// TIA Portal V19 export
FUNCTION "KP8 Interface" : Void   // FC3, LAD
{ S7_Optimized_Access := 'TRUE' }
// stored: SetENOAutomatically false
   VAR_TEMP
      RetVal : Int;
   END_VAR
   VAR_TEMP   // added for the SCL form of the ladder/FBD networks
      _w1 : Bool;
      _w2 : Bool;
   END_VAR
BEGIN

REGION Network 1: Turn all buttons white by default
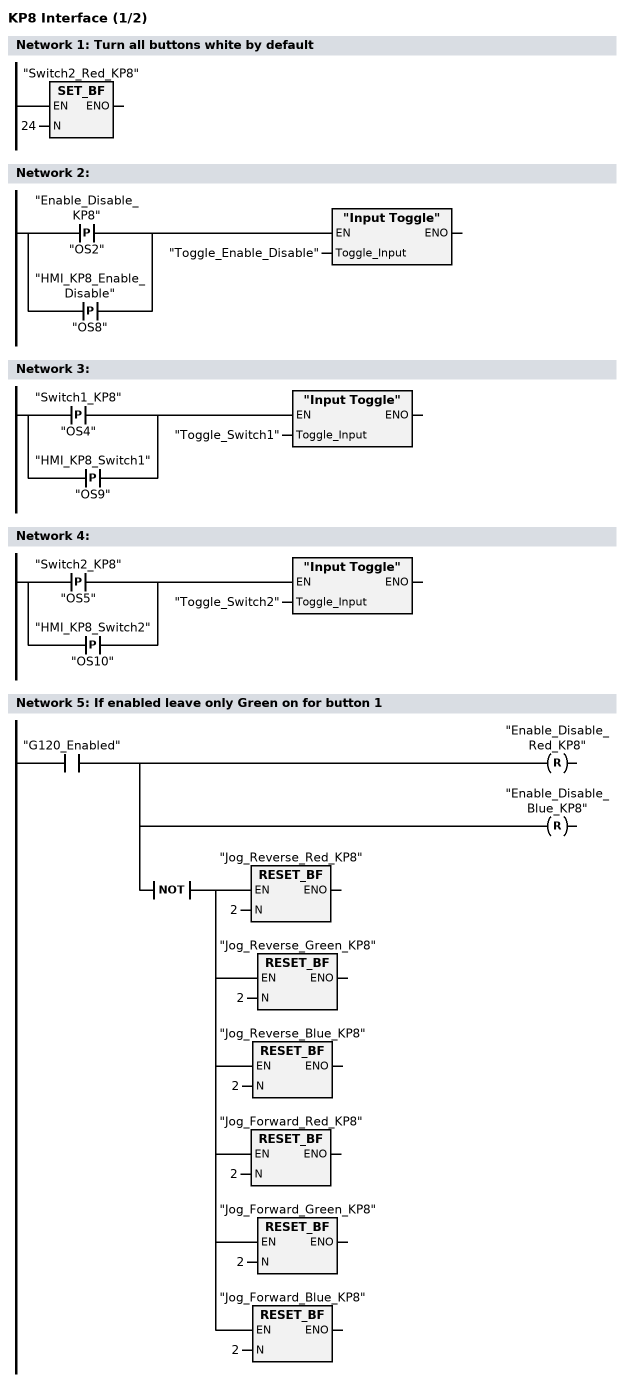
   // no SCL statement known for SBitfield: written as a call
   SET_BF(operand := "Switch2_Red_KP8", n := 24);
END_REGION

REGION Network 2
   RUNG wire#powerrail
      P_Contact(operand := "Enable_Disable_KP8", bit := "OS2")
      wire#w1
      "Input Toggle"(Toggle_Input := "Toggle_Enable_Disable")
   END_RUNG
   RUNG wire#powerrail
      P_Contact(operand := "HMI_KP8_Enable_Disable", bit := "OS8")
   END_RUNG wire#w1
   // the same network as SCL:
   #_w1 := "Enable_Disable_KP8" AND NOT "OS2";   // rising edge of "Enable_Disable_KP8"
   "OS2" := "Enable_Disable_KP8";
   #_w2 := "HMI_KP8_Enable_Disable" AND NOT "OS8";   // rising edge of "HMI_KP8_Enable_Disable"
   "OS8" := "HMI_KP8_Enable_Disable";
   IF #_w1 OR #_w2 THEN "Input Toggle"(Toggle_Input := "Toggle_Enable_Disable"); END_IF;
END_REGION

REGION Network 3
   RUNG wire#powerrail
      P_Contact(operand := "Switch1_KP8", bit := "OS4")
      wire#w1
      "Input Toggle"(Toggle_Input := "Toggle_Switch1")
   END_RUNG
   RUNG wire#powerrail
      P_Contact(operand := "HMI_KP8_Switch1", bit := "OS9")
   END_RUNG wire#w1
   // the same network as SCL:
   #_w1 := "Switch1_KP8" AND NOT "OS4";   // rising edge of "Switch1_KP8"
   "OS4" := "Switch1_KP8";
   #_w2 := "HMI_KP8_Switch1" AND NOT "OS9";   // rising edge of "HMI_KP8_Switch1"
   "OS9" := "HMI_KP8_Switch1";
   IF #_w1 OR #_w2 THEN "Input Toggle"(Toggle_Input := "Toggle_Switch1"); END_IF;
END_REGION

REGION Network 4
   RUNG wire#powerrail
      P_Contact(operand := "Switch2_KP8", bit := "OS5")
      wire#w1
      "Input Toggle"(Toggle_Input := "Toggle_Switch2")
   END_RUNG
   RUNG wire#powerrail
      P_Contact(operand := "HMI_KP8_Switch2", bit := "OS10")
   END_RUNG wire#w1
   // the same network as SCL:
   #_w1 := "Switch2_KP8" AND NOT "OS5";   // rising edge of "Switch2_KP8"
   "OS5" := "Switch2_KP8";
   #_w2 := "HMI_KP8_Switch2" AND NOT "OS10";   // rising edge of "HMI_KP8_Switch2"
   "OS10" := "HMI_KP8_Switch2";
   IF #_w1 OR #_w2 THEN "Input Toggle"(Toggle_Input := "Toggle_Switch2"); END_IF;
END_REGION

REGION Network 5: If enabled leave only Green on for button 1
   // no SCL statement known for RBitfield: written as a call
   IF "G120_Enabled" THEN
       "Enable_Disable_Red_KP8" := FALSE;
       "Enable_Disable_Blue_KP8" := FALSE;
   END_IF;
   #_w1 := NOT "G120_Enabled";
   IF #_w1 THEN
       RESET_BF(operand := "Jog_Reverse_Red_KP8", n := 2);
       RESET_BF(operand := "Jog_Reverse_Green_KP8", n := 2);
       RESET_BF(operand := "Jog_Reverse_Blue_KP8", n := 2);
       RESET_BF(operand := "Jog_Forward_Red_KP8", n := 2);
       RESET_BF(operand := "Jog_Forward_Green_KP8", n := 2);
       RESET_BF(operand := "Jog_Forward_Blue_KP8", n := 2);
   END_IF;
END_REGION

REGION Network 6: If there is an error flash red for button 5 by turning off other 2 leds
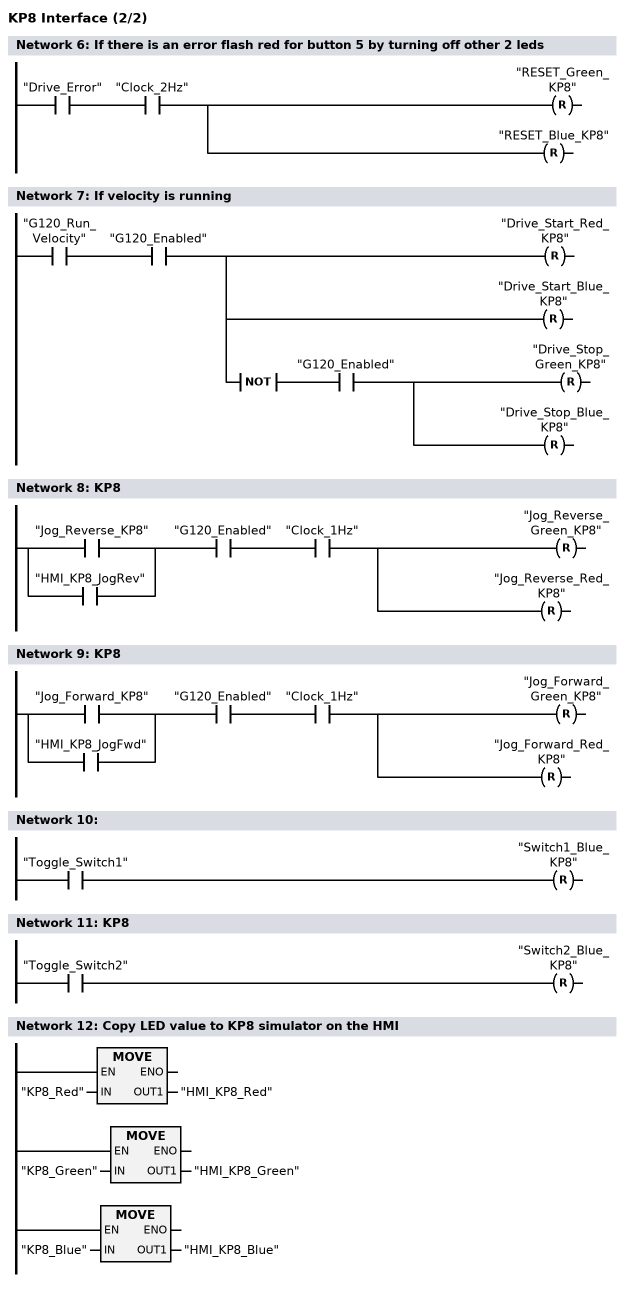
   RUNG wire#powerrail
      Contact( "Drive_Error" )
      Contact( "Clock_2Hz" )
      wire#w1
      R_Coil( "RESET_Green_KP8" )
   END_RUNG
   RUNG wire#w1
      R_Coil( "RESET_Blue_KP8" )
   END_RUNG
   // the same network as SCL:
   IF "Drive_Error" AND "Clock_2Hz" THEN
       "RESET_Green_KP8" := FALSE;
       "RESET_Blue_KP8" := FALSE;
   END_IF;
END_REGION

REGION Network 7: If velocity is running
   RUNG wire#powerrail
      Contact( "G120_Run_Velocity" )
      Contact( "G120_Enabled" )
      wire#w1
      R_Coil( "Drive_Start_Red_KP8" )
   END_RUNG
   RUNG wire#w1
      R_Coil( "Drive_Start_Blue_KP8" )
   END_RUNG
   RUNG wire#w1
      Not()
      Contact( "G120_Enabled" )
      wire#w2
      R_Coil( "Drive_Stop_Green_KP8" )
   END_RUNG
   RUNG wire#w2
      R_Coil( "Drive_Stop_Blue_KP8" )
   END_RUNG
   // the same network as SCL:
   #_w1 := "G120_Run_Velocity" AND "G120_Enabled";
   IF #_w1 THEN
       "Drive_Start_Red_KP8" := FALSE;
       "Drive_Start_Blue_KP8" := FALSE;
   END_IF;
   IF NOT #_w1 AND "G120_Enabled" THEN
       "Drive_Stop_Green_KP8" := FALSE;
       "Drive_Stop_Blue_KP8" := FALSE;
   END_IF;
END_REGION

REGION Network 8: KP8
   RUNG wire#powerrail
      Contact( "Jog_Reverse_KP8" )
      wire#w1
      Contact( "G120_Enabled" )
      Contact( "Clock_1Hz" )
      wire#w2
      R_Coil( "Jog_Reverse_Green_KP8" )
   END_RUNG
   RUNG wire#powerrail
      Contact( "HMI_KP8_JogRev" )
   END_RUNG wire#w1
   RUNG wire#w2
      R_Coil( "Jog_Reverse_Red_KP8" )
   END_RUNG
   // the same network as SCL:
   IF ("Jog_Reverse_KP8" OR "HMI_KP8_JogRev") AND "G120_Enabled" AND "Clock_1Hz" THEN
       "Jog_Reverse_Green_KP8" := FALSE;
       "Jog_Reverse_Red_KP8" := FALSE;
   END_IF;
END_REGION

REGION Network 9: KP8
   RUNG wire#powerrail
      Contact( "Jog_Forward_KP8" )
      wire#w1
      Contact( "G120_Enabled" )
      Contact( "Clock_1Hz" )
      wire#w2
      R_Coil( "Jog_Forward_Green_KP8" )
   END_RUNG
   RUNG wire#powerrail
      Contact( "HMI_KP8_JogFwd" )
   END_RUNG wire#w1
   RUNG wire#w2
      R_Coil( "Jog_Forward_Red_KP8" )
   END_RUNG
   // the same network as SCL:
   IF ("Jog_Forward_KP8" OR "HMI_KP8_JogFwd") AND "G120_Enabled" AND "Clock_1Hz" THEN
       "Jog_Forward_Green_KP8" := FALSE;
       "Jog_Forward_Red_KP8" := FALSE;
   END_IF;
END_REGION

REGION Network 10
   RUNG wire#powerrail
      Contact( "Toggle_Switch1" )
      R_Coil( "Switch1_Blue_KP8" )
   END_RUNG
   // the same network as SCL:
   IF "Toggle_Switch1" THEN "Switch1_Blue_KP8" := FALSE; END_IF;
END_REGION

REGION Network 11: KP8
   RUNG wire#powerrail
      Contact( "Toggle_Switch2" )
      R_Coil( "Switch2_Blue_KP8" )
   END_RUNG
   // the same network as SCL:
   IF "Toggle_Switch2" THEN "Switch2_Blue_KP8" := FALSE; END_IF;
END_REGION

REGION Network 12: Copy LED value to KP8 simulator on the HMI
   RUNG wire#powerrail
      Move(in := "KP8_Red", out1 => "HMI_KP8_Red")
   END_RUNG
   RUNG wire#powerrail
      Move(in := "KP8_Green", out1 => "HMI_KP8_Green")
   END_RUNG
   RUNG wire#powerrail
      Move(in := "KP8_Blue", out1 => "HMI_KP8_Blue")
   END_RUNG
   // the same network as SCL:
   "HMI_KP8_Red" := "KP8_Red";
   "HMI_KP8_Green" := "KP8_Green";
   "HMI_KP8_Blue" := "KP8_Blue";
END_REGION
END_FUNCTION
